(* PLC project MotionTest1, Higen MCL 1 *)
(* stored: creationDateTime 2012-01-06T15:20:13, modificationDateTime 2012-10-07T23:31:08 *)

FUNCTION_BLOCK wxgetval
  VAR
    getpy : python_gear;
    latch : SR;
  END_VAR
  VAR_INPUT
    name : STRING;
  END_VAR
  VAR_OUTPUT
    val : BOOL;
  END_VAR
  VAR  (* added by the conversion: wires and edge detectors of the diagram *)
    _EQ41_ENO : BOOL;
    _EQ41_OUT : BOOL;
    _EQ3_ENO : BOOL;
    _EQ3_OUT : BOOL;
  END_VAR

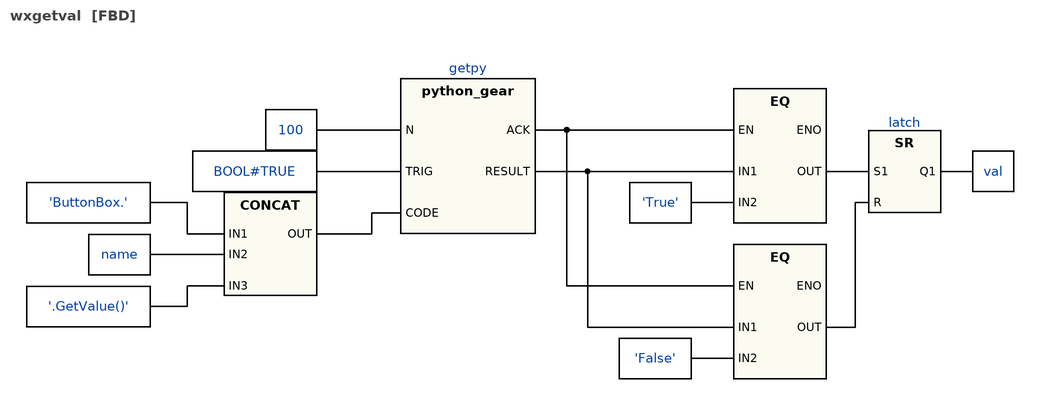
(* FBD diagram, written out as Structured Text *)
getpy(N := 100, TRIG := BOOL#TRUE, CODE := CONCAT('ButtonBox.', name, '.GetValue()'));
_EQ41_OUT := EQ(EN := getpy.ACK, IN1 := getpy.RESULT, IN2 := 'True', ENO => _EQ41_ENO);
_EQ3_OUT := EQ(EN := getpy.ACK, IN1 := getpy.RESULT, IN2 := 'False', ENO => _EQ3_ENO);
latch(S1 := _EQ41_OUT, R := _EQ3_OUT);
val := latch.Q1;
END_FUNCTION_BLOCK

PROGRAM main
  VAR
    Done : BOOL;
    Axis : AXIS_REF;
    moveA : MC_MoveAbsolute;
    switch : MC_Power;
    readpos : MC_ReadActualPosition;
    Pn : LREAL;
    Vn : LREAL;
    setpos : MC_SetPosition;
    readspeed : MC_ReadParameter;
    moveB : MC_Stop;
    sim : MC_Sim;
    bt1 : wxgetval;
    Block1 : wxgetval;
    Block2 : wxgetval;
    stat : MC_ReadStatus;
    Block3 : wxgetval;
    rset : MC_Reset;
    Block4 : wxgetval;
    p1 : MC_WriteParameter;
    Block5 : MC_WriteParameter;
    Block6 : wxgetval;
  END_VAR

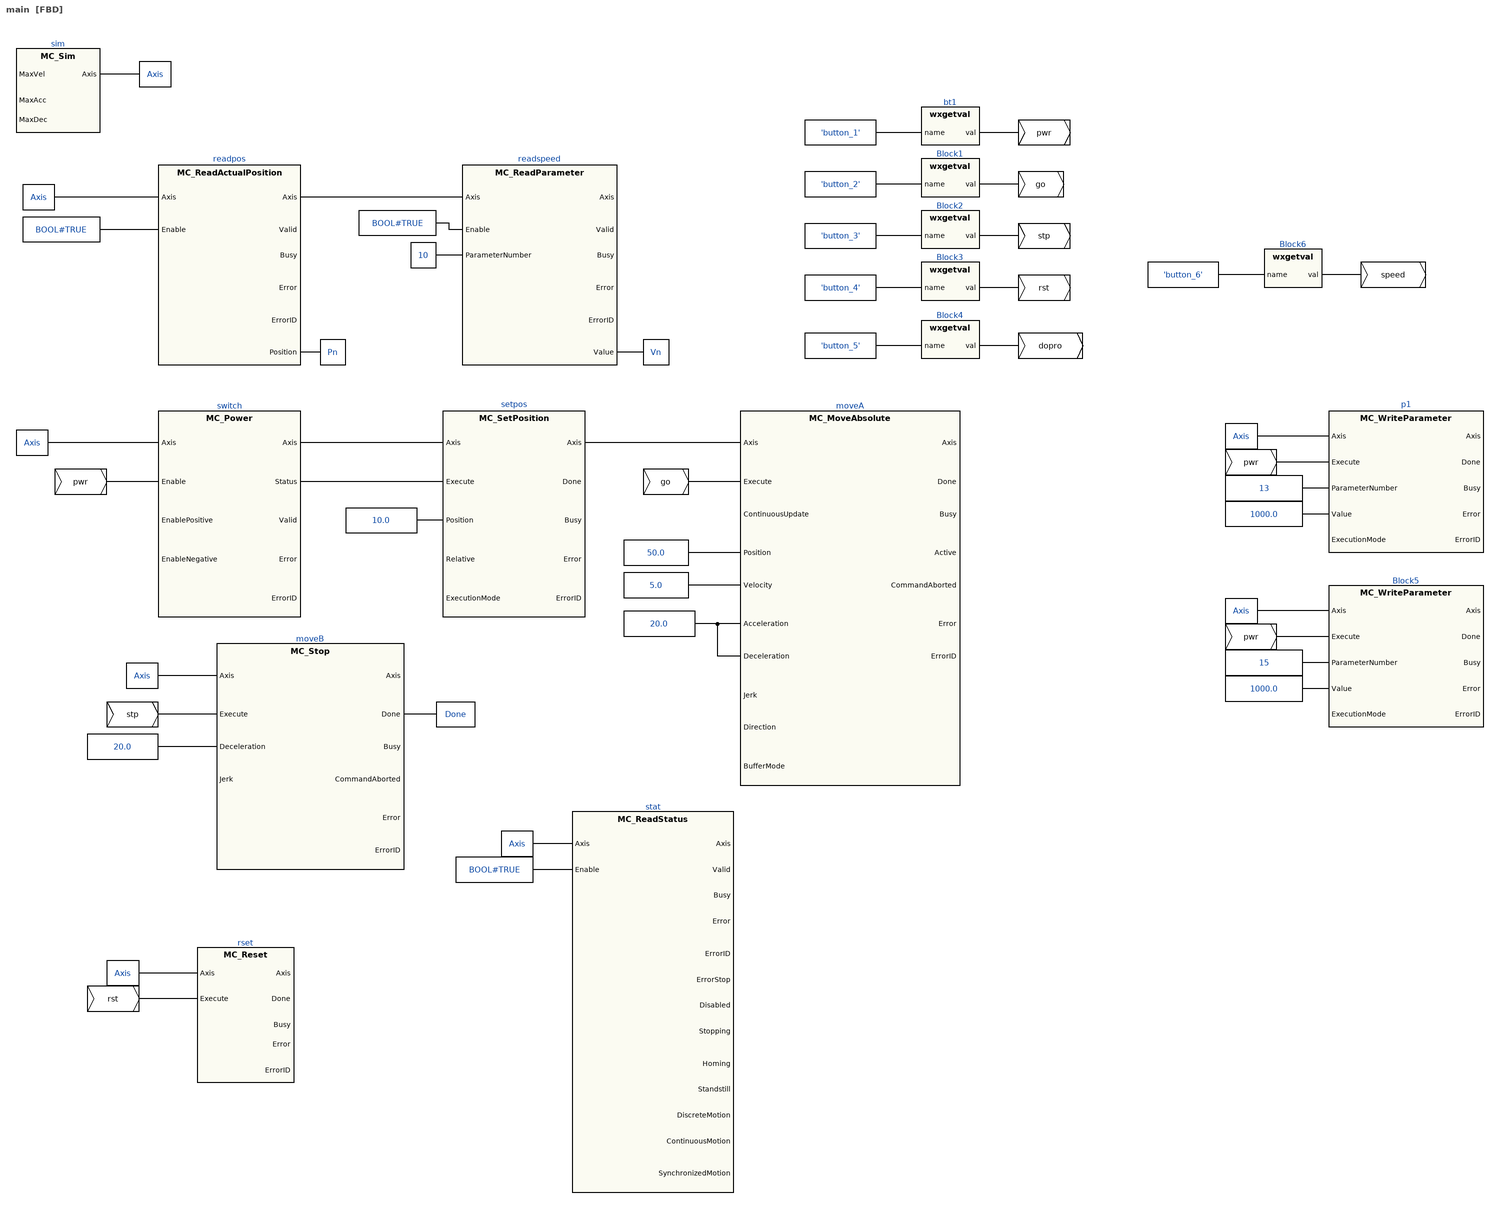
(* FBD diagram, written out as Structured Text *)
sim();
Axis := sim.Axis;
readpos(Axis := Axis, Enable := BOOL#TRUE);
Pn := readpos.Position;
readspeed(Axis := readpos.Axis, Enable := BOOL#TRUE, ParameterNumber := 10);
Vn := readspeed.Value;
Block2(name := 'button_3');
moveB(Axis := Axis, Execute := Block2.val, Deceleration := 20.0);
Done := moveB.Done;
bt1(name := 'button_1');
Block1(name := 'button_2');
Block6(name := 'button_6');
Block3(name := 'button_4');
Block4(name := 'button_5');
switch(Axis := Axis, Enable := bt1.val);
setpos(Axis := switch.Axis, Execute := switch.Status, Position := 10.0);
moveA(Axis := setpos.Axis, Execute := Block1.val, Position := 50.0, Velocity := 5.0, Acceleration := 20.0, Deceleration := 20.0);
p1(Axis := Axis, Execute := bt1.val, ParameterNumber := 13, Value := 1000.0);
Block5(Axis := Axis, Execute := bt1.val, ParameterNumber := 15, Value := 1000.0);
stat(Axis := Axis, Enable := BOOL#TRUE);
rset(Axis := Axis, Execute := Block3.val);
END_PROGRAM

CONFIGURATION conf
  RESOURCE res ON PLC
    TASK milisecond(INTERVAL := T#1ms, PRIORITY := 0);
    PROGRAM maininstance WITH milisecond : main;
  END_RESOURCE
END_CONFIGURATION
